// TIA Portal V20 export
FUNCTION "03 T10 LANT Aux" : Void   // FC1393, LAD
TITLE = AUXILIARIES
{ S7_Optimized_Access := 'TRUE' }
// stored: AutoNumber false, SetENOAutomatically false
   VAR_TEMP
      Aux_OS : Bool;
      Aux_sup : Real;
      Aux_inf : Real;
      Aux_DInt : DInt;
      Aux_Real : Real;
   END_VAR
   VAR CONSTANT
      "Max differenza L tubi" : Real := 500.0;
   END_VAR
   VAR_TEMP   // added for the SCL form of the ladder/FBD networks
      _w1 : Bool;
      _w2 : Bool;
      _w3 : Bool;
   END_VAR
BEGIN

REGION Network 1: =========== MEMORIES ===========
END_REGION

REGION Network 2: Piece presence
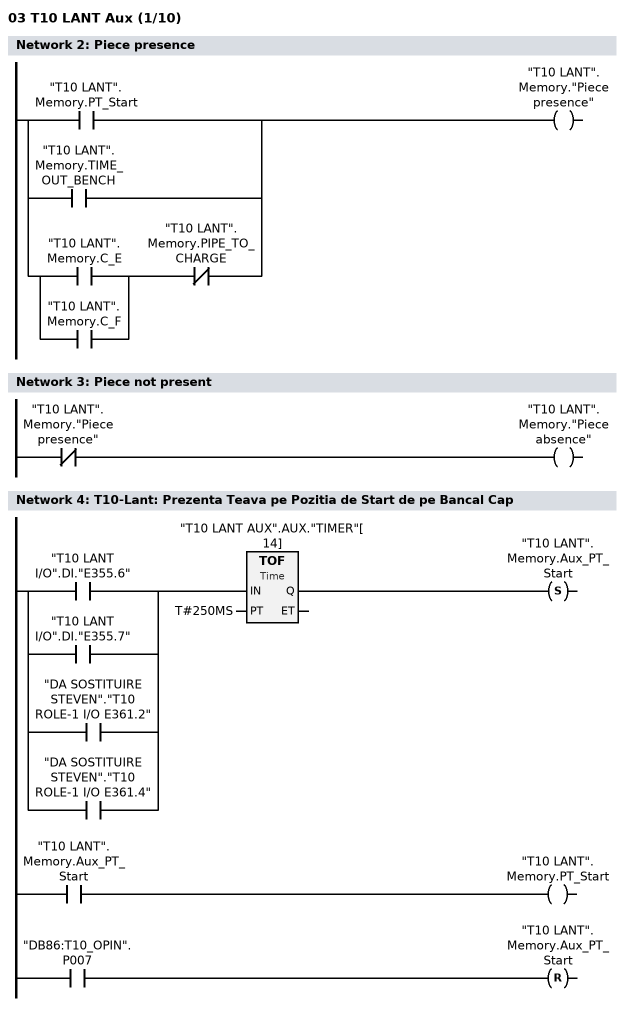
   RUNG wire#powerrail
      Contact( "T10 LANT".Memory.PT_Start )
      wire#w1
      Coil( "T10 LANT".Memory."Piece presence" )
   END_RUNG
   RUNG wire#powerrail
      Contact( "T10 LANT".Memory.TIME_OUT_BENCH )
   END_RUNG wire#w1
   RUNG wire#powerrail
      Contact( "T10 LANT".Memory.C_E )
      wire#w2
      I_Contact( "T10 LANT".Memory.PIPE_TO_CHARGE )
   END_RUNG wire#w1
   RUNG wire#powerrail
      Contact( "T10 LANT".Memory.C_F )
   END_RUNG wire#w2
   // the same network as SCL:
   "T10 LANT".Memory."Piece presence" := "T10 LANT".Memory.PT_Start OR "T10 LANT".Memory.TIME_OUT_BENCH OR (("T10 LANT".Memory.C_E OR "T10 LANT".Memory.C_F) AND NOT "T10 LANT".Memory.PIPE_TO_CHARGE);
END_REGION

REGION Network 3: Piece not present
   RUNG wire#powerrail
      I_Contact( "T10 LANT".Memory."Piece presence" )
      Coil( "T10 LANT".Memory."Piece absence" )
   END_RUNG
   // the same network as SCL:
   "T10 LANT".Memory."Piece absence" := NOT "T10 LANT".Memory."Piece presence";
END_REGION

REGION Network 4: T10-Lant: Prezenta Teava pe Pozitia de Start de pe Bancal Cap
   RUNG wire#powerrail
      Contact( "T10 LANT I/O".DI."E355.6" )
      wire#w1
      { S7_Templates := "time_type := Time" } "T10 LANT AUX".AUX."TIMER"[14].TOF(pt := T#250MS, et =>)
      S_Coil( "T10 LANT".Memory.Aux_PT_Start )
   END_RUNG
   RUNG wire#powerrail
      Contact( "T10 LANT I/O".DI."E355.7" )
   END_RUNG wire#w1
   RUNG wire#powerrail
      Contact( "DA SOSTITUIRE STEVEN"."T10 ROLE-1 I/O E361.2" )
   END_RUNG wire#w1
   RUNG wire#powerrail
      Contact( "DA SOSTITUIRE STEVEN"."T10 ROLE-1 I/O E361.4" )
   END_RUNG wire#w1
   RUNG wire#powerrail
      Contact( "T10 LANT".Memory.Aux_PT_Start )
      Coil( "T10 LANT".Memory.PT_Start )
   END_RUNG
   RUNG wire#powerrail
      Contact( "DB86:T10_OPIN".P007 )
      R_Coil( "T10 LANT".Memory.Aux_PT_Start )
   END_RUNG
   // the same network as SCL:
   "T10 LANT AUX".AUX."TIMER"[14].TOF(IN := "T10 LANT I/O".DI."E355.6" OR "T10 LANT I/O".DI."E355.7" OR "DA SOSTITUIRE STEVEN"."T10 ROLE-1 I/O E361.2" OR "DA SOSTITUIRE STEVEN"."T10 ROLE-1 I/O E361.4",
                           PT := T#250MS);
   IF "T10 LANT AUX".AUX."TIMER"[14].Q THEN "T10 LANT".Memory.Aux_PT_Start := TRUE; END_IF;
   "T10 LANT".Memory.PT_Start := "T10 LANT".Memory.Aux_PT_Start;
   IF "DB86:T10_OPIN".P007 THEN "T10 LANT".Memory.Aux_PT_Start := FALSE; END_IF;
END_REGION

REGION Network 5: T10-Lant: Prezenta Teava pe Pozitia de 'Incetinire' de pe Bancal
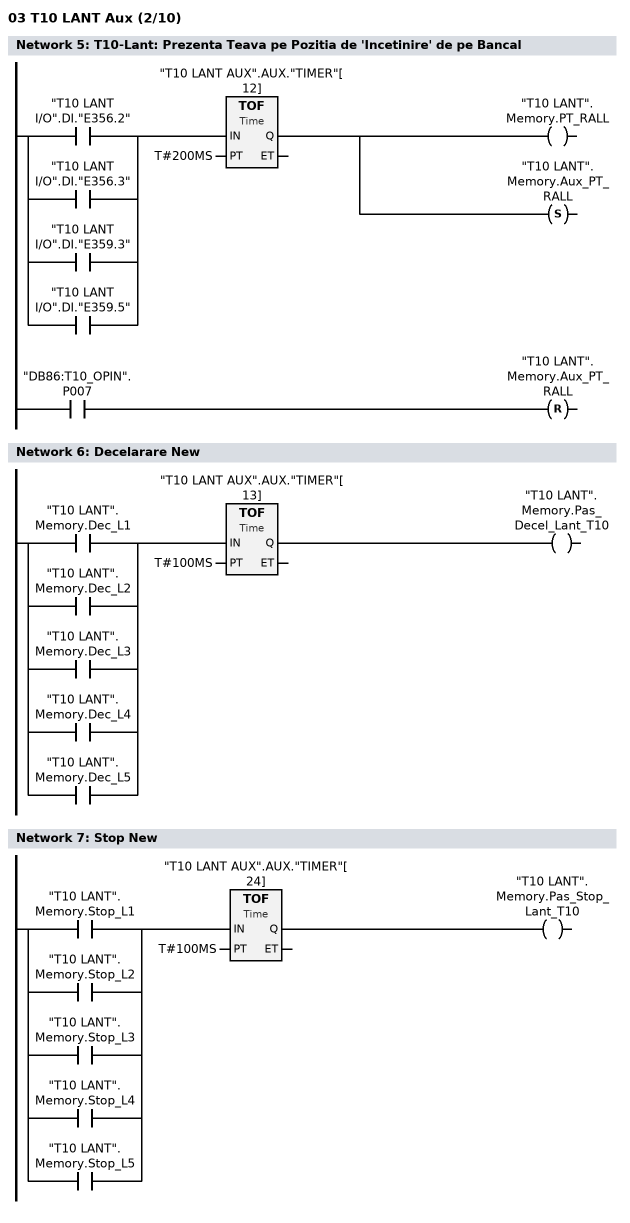
   RUNG wire#powerrail
      Contact( "T10 LANT I/O".DI."E356.2" )
      wire#w1
      { S7_Templates := "time_type := Time" } "T10 LANT AUX".AUX."TIMER"[12].TOF(pt := T#200MS, et =>)
      wire#w2
      Coil( "T10 LANT".Memory.PT_RALL )
   END_RUNG
   RUNG wire#powerrail
      Contact( "T10 LANT I/O".DI."E356.3" )
   END_RUNG wire#w1
   RUNG wire#powerrail
      Contact( "T10 LANT I/O".DI."E359.3" )
   END_RUNG wire#w1
   RUNG wire#powerrail
      Contact( "T10 LANT I/O".DI."E359.5" )
   END_RUNG wire#w1
   RUNG wire#w2
      S_Coil( "T10 LANT".Memory.Aux_PT_RALL )
   END_RUNG
   RUNG wire#powerrail
      Contact( "DB86:T10_OPIN".P007 )
      R_Coil( "T10 LANT".Memory.Aux_PT_RALL )
   END_RUNG
   // the same network as SCL:
   "T10 LANT AUX".AUX."TIMER"[12].TOF(IN := "T10 LANT I/O".DI."E356.2" OR "T10 LANT I/O".DI."E356.3" OR "T10 LANT I/O".DI."E359.3" OR "T10 LANT I/O".DI."E359.5",
                           PT := T#200MS);
   "T10 LANT".Memory.PT_RALL := "T10 LANT AUX".AUX."TIMER"[12].Q;
   IF "T10 LANT AUX".AUX."TIMER"[12].Q THEN "T10 LANT".Memory.Aux_PT_RALL := TRUE; END_IF;
   IF "DB86:T10_OPIN".P007 THEN "T10 LANT".Memory.Aux_PT_RALL := FALSE; END_IF;
END_REGION

REGION Network 6: Decelarare New
   RUNG wire#powerrail
      Contact( "T10 LANT".Memory.Dec_L1 )
      wire#w1
      { S7_Templates := "time_type := Time" } "T10 LANT AUX".AUX."TIMER"[13].TOF(pt := T#100MS, et =>)
      Coil( "T10 LANT".Memory.Pas_Decel_Lant_T10 )
   END_RUNG
   RUNG wire#powerrail
      Contact( "T10 LANT".Memory.Dec_L2 )
   END_RUNG wire#w1
   RUNG wire#powerrail
      Contact( "T10 LANT".Memory.Dec_L3 )
   END_RUNG wire#w1
   RUNG wire#powerrail
      Contact( "T10 LANT".Memory.Dec_L4 )
   END_RUNG wire#w1
   RUNG wire#powerrail
      Contact( "T10 LANT".Memory.Dec_L5 )
   END_RUNG wire#w1
   // the same network as SCL:
   "T10 LANT AUX".AUX."TIMER"[13].TOF(IN := "T10 LANT".Memory.Dec_L1 OR "T10 LANT".Memory.Dec_L2 OR "T10 LANT".Memory.Dec_L3 OR "T10 LANT".Memory.Dec_L4 OR "T10 LANT".Memory.Dec_L5,
                           PT := T#100MS);
   "T10 LANT".Memory.Pas_Decel_Lant_T10 := "T10 LANT AUX".AUX."TIMER"[13].Q;
END_REGION

REGION Network 7: Stop New
   RUNG wire#powerrail
      Contact( "T10 LANT".Memory.Stop_L1 )
      wire#w1
      { S7_Templates := "time_type := Time" } "T10 LANT AUX".AUX."TIMER"[24].TOF(pt := T#100MS, et =>)
      Coil( "T10 LANT".Memory.Pas_Stop_Lant_T10 )
   END_RUNG
   RUNG wire#powerrail
      Contact( "T10 LANT".Memory.Stop_L2 )
   END_RUNG wire#w1
   RUNG wire#powerrail
      Contact( "T10 LANT".Memory.Stop_L3 )
   END_RUNG wire#w1
   RUNG wire#powerrail
      Contact( "T10 LANT".Memory.Stop_L4 )
   END_RUNG wire#w1
   RUNG wire#powerrail
      Contact( "T10 LANT".Memory.Stop_L5 )
   END_RUNG wire#w1
   // the same network as SCL:
   "T10 LANT AUX".AUX."TIMER"[24].TOF(IN := "T10 LANT".Memory.Stop_L1 OR "T10 LANT".Memory.Stop_L2 OR "T10 LANT".Memory.Stop_L3 OR "T10 LANT".Memory.Stop_L4 OR "T10 LANT".Memory.Stop_L5,
                           PT := T#100MS);
   "T10 LANT".Memory.Pas_Stop_Lant_T10 := "T10 LANT AUX".AUX."TIMER"[24].Q;
END_REGION

REGION Network 8: T10-Lant: LAnt in Pozitia 'Pas'
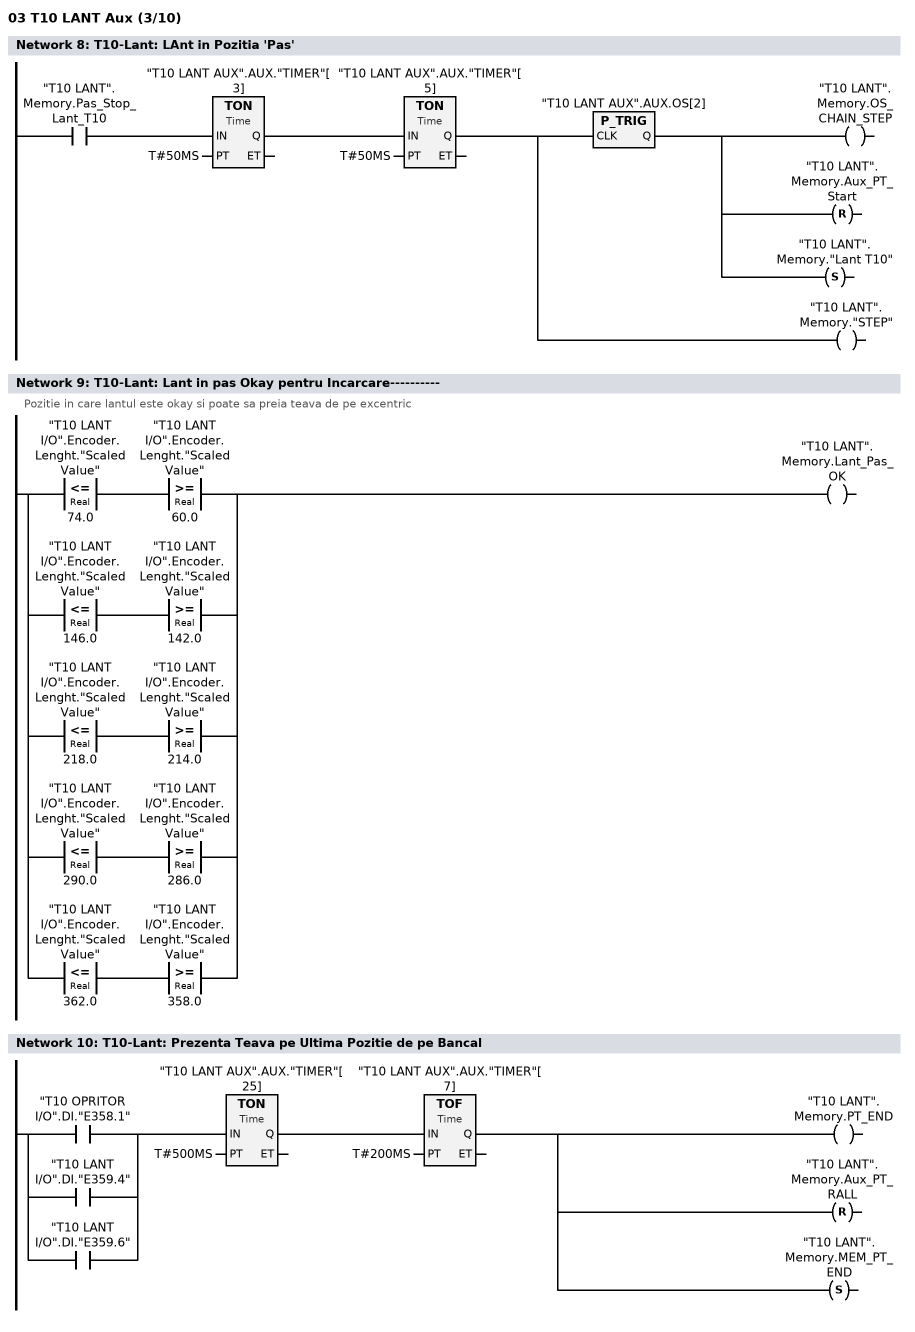
   RUNG wire#powerrail
      Contact( "T10 LANT".Memory.Pas_Stop_Lant_T10 )
      { S7_Templates := "time_type := Time" } "T10 LANT AUX".AUX."TIMER"[3].TON(pt := T#50MS, et =>)
      { S7_Templates := "time_type := Time" } "T10 LANT AUX".AUX."TIMER"[5].TON(pt := T#50MS, et =>)
      wire#w1
      P_Trig( "T10 LANT AUX".AUX.OS[2] )
      wire#w2
      Coil( "T10 LANT".Memory.OS_CHAIN_STEP )
   END_RUNG
   RUNG wire#w2
      R_Coil( "T10 LANT".Memory.Aux_PT_Start )
   END_RUNG
   RUNG wire#w2
      S_Coil( "T10 LANT".Memory."Lant T10" )
   END_RUNG
   RUNG wire#w1
      Coil( "T10 LANT".Memory."STEP" )
   END_RUNG
   // the same network as SCL:
   "T10 LANT AUX".AUX."TIMER"[3].TON(IN := "T10 LANT".Memory.Pas_Stop_Lant_T10, PT := T#50MS);
   "T10 LANT AUX".AUX."TIMER"[5].TON(IN := "T10 LANT AUX".AUX."TIMER"[3].Q, PT := T#50MS);
   #_w1 := "T10 LANT AUX".AUX."TIMER"[5].Q AND NOT "T10 LANT AUX".AUX.OS[2];   // rising edge
   "T10 LANT AUX".AUX.OS[2] := "T10 LANT AUX".AUX."TIMER"[5].Q;
   "T10 LANT".Memory.OS_CHAIN_STEP := #_w1;
   IF #_w1 THEN
       "T10 LANT".Memory.Aux_PT_Start := FALSE;
       "T10 LANT".Memory."Lant T10" := TRUE;
   END_IF;
   "T10 LANT".Memory."STEP" := "T10 LANT AUX".AUX."TIMER"[5].Q;
END_REGION

REGION Network 9: T10-Lant: Lant in pas Okay pentru Incarcare----------
   // Pozitie in care lantul este okay si poate sa preia teava de pe excentric
   RUNG wire#powerrail
      { S7_Templates := "SrcType := Real" } LE_Contact(in1 := "T10 LANT I/O".Encoder.Lenght."Scaled Value", in2 := 74.0)
      { S7_Templates := "SrcType := Real" } GE_Contact(in1 := "T10 LANT I/O".Encoder.Lenght."Scaled Value", in2 := 60.0)
      wire#w1
      Coil( "T10 LANT".Memory.Lant_Pas_OK )
   END_RUNG
   RUNG wire#powerrail
      { S7_Templates := "SrcType := Real" } LE_Contact(in1 := "T10 LANT I/O".Encoder.Lenght."Scaled Value", in2 := 146.0)
      { S7_Templates := "SrcType := Real" } GE_Contact(in1 := "T10 LANT I/O".Encoder.Lenght."Scaled Value", in2 := 142.0)
   END_RUNG wire#w1
   RUNG wire#powerrail
      { S7_Templates := "SrcType := Real" } LE_Contact(in1 := "T10 LANT I/O".Encoder.Lenght."Scaled Value", in2 := 218.0)
      { S7_Templates := "SrcType := Real" } GE_Contact(in1 := "T10 LANT I/O".Encoder.Lenght."Scaled Value", in2 := 214.0)
   END_RUNG wire#w1
   RUNG wire#powerrail
      { S7_Templates := "SrcType := Real" } LE_Contact(in1 := "T10 LANT I/O".Encoder.Lenght."Scaled Value", in2 := 290.0)
      { S7_Templates := "SrcType := Real" } GE_Contact(in1 := "T10 LANT I/O".Encoder.Lenght."Scaled Value", in2 := 286.0)
   END_RUNG wire#w1
   RUNG wire#powerrail
      { S7_Templates := "SrcType := Real" } LE_Contact(in1 := "T10 LANT I/O".Encoder.Lenght."Scaled Value", in2 := 362.0)
      { S7_Templates := "SrcType := Real" } GE_Contact(in1 := "T10 LANT I/O".Encoder.Lenght."Scaled Value", in2 := 358.0)
   END_RUNG wire#w1
   // the same network as SCL:
   "T10 LANT".Memory.Lant_Pas_OK := (("T10 LANT I/O".Encoder.Lenght."Scaled Value" <= 74.0) AND ("T10 LANT I/O".Encoder.Lenght."Scaled Value" >= 60.0)) OR (("T10 LANT I/O".Encoder.Lenght."Scaled Value" <= 146.0) AND ("T10 LANT I/O".Encoder.Lenght."Scaled Value" >= 142.0)) OR (("T10 LANT I/O".Encoder.Lenght."Scaled Value" <= 218.0) AND ("T10 LANT I/O".Encoder.Lenght."Scaled Value" >= 214.0)) OR (("T10 LANT I/O".Encoder.Lenght."Scaled Value" <= 290.0) AND ("T10 LANT I/O".Encoder.Lenght."Scaled Value" >= 286.0)) OR (("T10 LANT I/O".Encoder.Lenght."Scaled Value" <= 362.0) AND ("T10 LANT I/O".Encoder.Lenght."Scaled Value" >= 358.0));
END_REGION

REGION Network 10: T10-Lant: Prezenta Teava pe Ultima Pozitie de pe Bancal
   RUNG wire#powerrail
      Contact( "T10 OPRITOR I/O".DI."E358.1" )
      wire#w1
      { S7_Templates := "time_type := Time" } "T10 LANT AUX".AUX."TIMER"[25].TON(pt := T#500MS, et =>)
      { S7_Templates := "time_type := Time" } "T10 LANT AUX".AUX."TIMER"[7].TOF(pt := T#200MS, et =>)
      wire#w2
      Coil( "T10 LANT".Memory.PT_END )
   END_RUNG
   RUNG wire#powerrail
      Contact( "T10 LANT I/O".DI."E359.4" )
   END_RUNG wire#w1
   RUNG wire#powerrail
      Contact( "T10 LANT I/O".DI."E359.6" )
   END_RUNG wire#w1
   RUNG wire#w2
      R_Coil( "T10 LANT".Memory.Aux_PT_RALL )
   END_RUNG
   RUNG wire#w2
      S_Coil( "T10 LANT".Memory.MEM_PT_END )
   END_RUNG
   // the same network as SCL:
   "T10 LANT AUX".AUX."TIMER"[25].TON(IN := "T10 OPRITOR I/O".DI."E358.1" OR "T10 LANT I/O".DI."E359.4" OR "T10 LANT I/O".DI."E359.6",
                           PT := T#500MS);
   "T10 LANT AUX".AUX."TIMER"[7].TOF(IN := "T10 LANT AUX".AUX."TIMER"[25].Q, PT := T#200MS);
   "T10 LANT".Memory.PT_END := "T10 LANT AUX".AUX."TIMER"[7].Q;
   IF "T10 LANT AUX".AUX."TIMER"[7].Q THEN
       "T10 LANT".Memory.Aux_PT_RALL := FALSE;
       "T10 LANT".Memory.MEM_PT_END := TRUE;
   END_IF;
END_REGION

REGION Network 11: T10-Lant: TRK: Prezenta Teava pe Pozitia 'Incetinire' pe Bancal
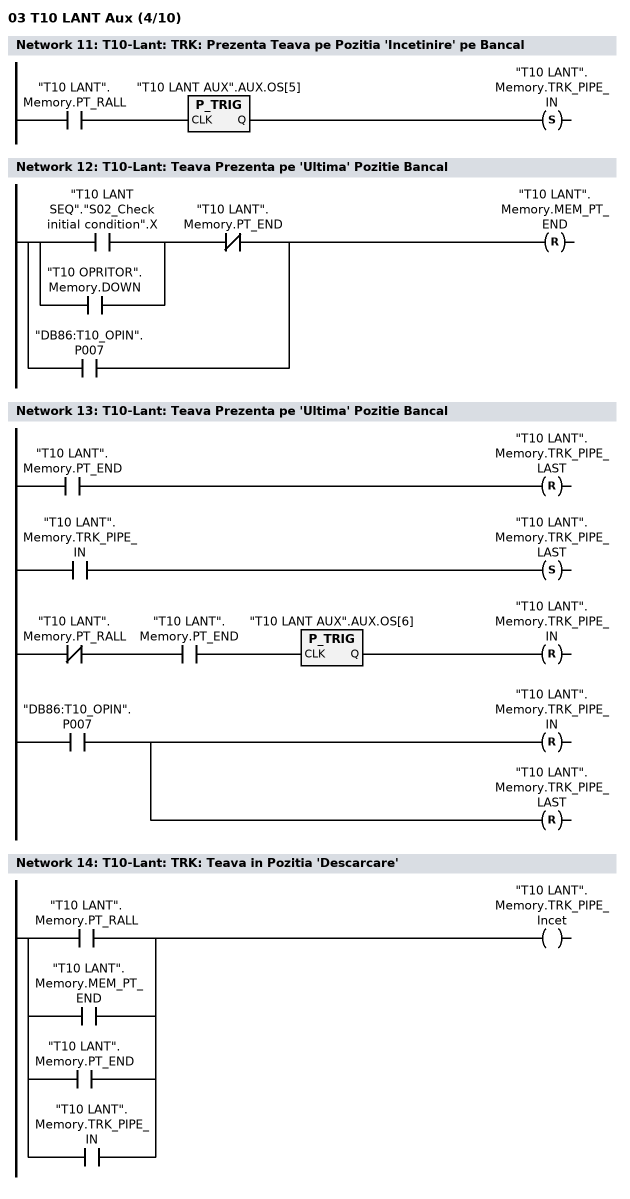
   RUNG wire#powerrail
      Contact( "T10 LANT".Memory.PT_RALL )
      P_Trig( "T10 LANT AUX".AUX.OS[5] )
      S_Coil( "T10 LANT".Memory.TRK_PIPE_IN )
   END_RUNG
   // the same network as SCL:
   #_w1 := "T10 LANT".Memory.PT_RALL AND NOT "T10 LANT AUX".AUX.OS[5];   // rising edge
   "T10 LANT AUX".AUX.OS[5] := "T10 LANT".Memory.PT_RALL;
   IF #_w1 THEN "T10 LANT".Memory.TRK_PIPE_IN := TRUE; END_IF;
END_REGION

REGION Network 12: T10-Lant: Teava Prezenta pe 'Ultima' Pozitie Bancal
   RUNG wire#powerrail
      Contact( "T10 LANT SEQ"."S02_Check initial condition".X )
      wire#w1
      I_Contact( "T10 LANT".Memory.PT_END )
      wire#w2
      R_Coil( "T10 LANT".Memory.MEM_PT_END )
   END_RUNG
   RUNG wire#powerrail
      Contact( "T10 OPRITOR".Memory.DOWN )
   END_RUNG wire#w1
   RUNG wire#powerrail
      Contact( "DB86:T10_OPIN".P007 )
   END_RUNG wire#w2
   // the same network as SCL:
   IF (("T10 LANT SEQ"."S02_Check initial condition".X OR "T10 OPRITOR".Memory.DOWN) AND NOT "T10 LANT".Memory.PT_END) OR "DB86:T10_OPIN".P007 THEN
       "T10 LANT".Memory.MEM_PT_END := FALSE;
   END_IF;
END_REGION

REGION Network 13: T10-Lant: Teava Prezenta pe 'Ultima' Pozitie Bancal
   RUNG wire#powerrail
      Contact( "T10 LANT".Memory.PT_END )
      R_Coil( "T10 LANT".Memory.TRK_PIPE_LAST )
   END_RUNG
   RUNG wire#powerrail
      Contact( "T10 LANT".Memory.TRK_PIPE_IN )
      S_Coil( "T10 LANT".Memory.TRK_PIPE_LAST )
   END_RUNG
   RUNG wire#powerrail
      I_Contact( "T10 LANT".Memory.PT_RALL )
      Contact( "T10 LANT".Memory.PT_END )
      P_Trig( "T10 LANT AUX".AUX.OS[6] )
      R_Coil( "T10 LANT".Memory.TRK_PIPE_IN )
   END_RUNG
   RUNG wire#powerrail
      Contact( "DB86:T10_OPIN".P007 )
      wire#w1
      R_Coil( "T10 LANT".Memory.TRK_PIPE_IN )
   END_RUNG
   RUNG wire#w1
      R_Coil( "T10 LANT".Memory.TRK_PIPE_LAST )
   END_RUNG
   // the same network as SCL:
   IF "T10 LANT".Memory.PT_END THEN "T10 LANT".Memory.TRK_PIPE_LAST := FALSE; END_IF;
   IF "T10 LANT".Memory.TRK_PIPE_IN THEN "T10 LANT".Memory.TRK_PIPE_LAST := TRUE; END_IF;
   #_w1 := NOT "T10 LANT".Memory.PT_RALL AND "T10 LANT".Memory.PT_END;
   #_w2 := #_w1 AND NOT "T10 LANT AUX".AUX.OS[6];   // rising edge
   "T10 LANT AUX".AUX.OS[6] := #_w1;
   IF #_w2 THEN "T10 LANT".Memory.TRK_PIPE_IN := FALSE; END_IF;
   IF "DB86:T10_OPIN".P007 THEN
       "T10 LANT".Memory.TRK_PIPE_IN := FALSE;
       "T10 LANT".Memory.TRK_PIPE_LAST := FALSE;
   END_IF;
END_REGION

REGION Network 14: T10-Lant: TRK: Teava in Pozitia 'Descarcare'
   RUNG wire#powerrail
      Contact( "T10 LANT".Memory.PT_RALL )
      wire#w1
      Coil( "T10 LANT".Memory.TRK_PIPE_Incet )
   END_RUNG
   RUNG wire#powerrail
      Contact( "T10 LANT".Memory.MEM_PT_END )
   END_RUNG wire#w1
   RUNG wire#powerrail
      Contact( "T10 LANT".Memory.PT_END )
   END_RUNG wire#w1
   RUNG wire#powerrail
      Contact( "T10 LANT".Memory.TRK_PIPE_IN )
   END_RUNG wire#w1
   // the same network as SCL:
   "T10 LANT".Memory.TRK_PIPE_Incet := "T10 LANT".Memory.PT_RALL OR "T10 LANT".Memory.MEM_PT_END OR "T10 LANT".Memory.PT_END OR "T10 LANT".Memory.TRK_PIPE_IN;
END_REGION

REGION Network 15: T10-Lant: Teava Pregatita pt. 'Incarcare'
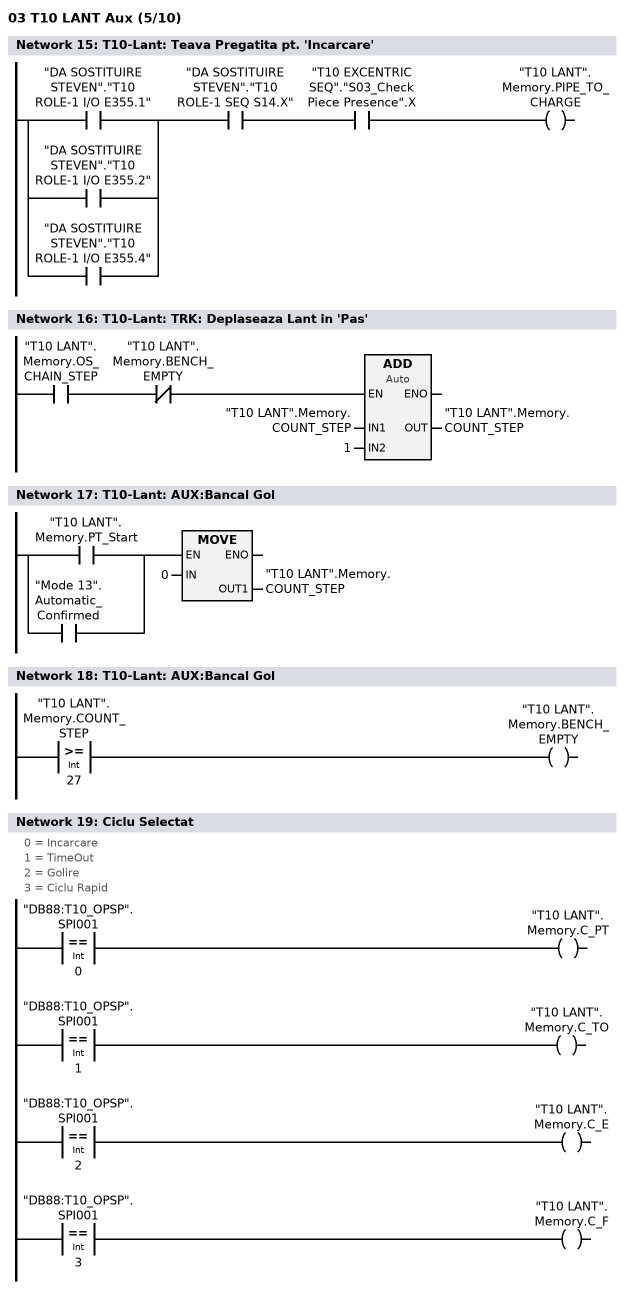
   RUNG wire#powerrail
      Contact( "DA SOSTITUIRE STEVEN"."T10 ROLE-1 I/O E355.1" )
      wire#w1
      Contact( "DA SOSTITUIRE STEVEN"."T10 ROLE-1 SEQ S14.X" )
      Contact( "T10 EXCENTRIC SEQ"."S03_Check Piece Presence".X )
      Coil( "T10 LANT".Memory.PIPE_TO_CHARGE )
   END_RUNG
   RUNG wire#powerrail
      Contact( "DA SOSTITUIRE STEVEN"."T10 ROLE-1 I/O E355.2" )
   END_RUNG wire#w1
   RUNG wire#powerrail
      Contact( "DA SOSTITUIRE STEVEN"."T10 ROLE-1 I/O E355.4" )
   END_RUNG wire#w1
   // the same network as SCL:
   "T10 LANT".Memory.PIPE_TO_CHARGE := ("DA SOSTITUIRE STEVEN"."T10 ROLE-1 I/O E355.1" OR "DA SOSTITUIRE STEVEN"."T10 ROLE-1 I/O E355.2" OR "DA SOSTITUIRE STEVEN"."T10 ROLE-1 I/O E355.4") AND "DA SOSTITUIRE STEVEN"."T10 ROLE-1 SEQ S14.X" AND "T10 EXCENTRIC SEQ"."S03_Check Piece Presence".X;
END_REGION

REGION Network 16: T10-Lant: TRK: Deplaseaza Lant in 'Pas'
   RUNG wire#powerrail
      Contact( "T10 LANT".Memory.OS_CHAIN_STEP )
      I_Contact( "T10 LANT".Memory.BENCH_EMPTY )
      Add(in1 := "T10 LANT".Memory.COUNT_STEP, in2 := 1, out => "T10 LANT".Memory.COUNT_STEP)
   END_RUNG
   // the same network as SCL:
   IF "T10 LANT".Memory.OS_CHAIN_STEP AND NOT "T10 LANT".Memory.BENCH_EMPTY THEN
       "T10 LANT".Memory.COUNT_STEP := "T10 LANT".Memory.COUNT_STEP + 1;
   END_IF;
END_REGION

REGION Network 17: T10-Lant: AUX:Bancal Gol
   RUNG wire#powerrail
      Contact( "T10 LANT".Memory.PT_Start )
      wire#w1
      Move(in := 0, out1 => "T10 LANT".Memory.COUNT_STEP)
   END_RUNG
   RUNG wire#powerrail
      Contact( "Mode 13".Automatic_Confirmed )
   END_RUNG wire#w1
   // the same network as SCL:
   IF "T10 LANT".Memory.PT_Start OR "Mode 13".Automatic_Confirmed THEN
       "T10 LANT".Memory.COUNT_STEP := 0;
   END_IF;
END_REGION

REGION Network 18: T10-Lant: AUX:Bancal Gol
   RUNG wire#powerrail
      { S7_Templates := "SrcType := Int" } GE_Contact(in1 := "T10 LANT".Memory.COUNT_STEP, in2 := 27)
      Coil( "T10 LANT".Memory.BENCH_EMPTY )
   END_RUNG
   // the same network as SCL:
   "T10 LANT".Memory.BENCH_EMPTY := "T10 LANT".Memory.COUNT_STEP >= 27;
END_REGION

REGION Network 19: Ciclu Selectat
   // 0 = Incarcare 
   // 1 = TimeOut
   // 2 = Golire
   // 3 = Ciclu Rapid
   RUNG wire#powerrail
      { S7_Templates := "SrcType := Int" } EQ_Contact(in1 := "DB88:T10_OPSP".SPI001, in2 := 0)
      Coil( "T10 LANT".Memory.C_PT )
   END_RUNG
   RUNG wire#powerrail
      { S7_Templates := "SrcType := Int" } EQ_Contact(in1 := "DB88:T10_OPSP".SPI001, in2 := 1)
      Coil( "T10 LANT".Memory.C_TO )
   END_RUNG
   RUNG wire#powerrail
      { S7_Templates := "SrcType := Int" } EQ_Contact(in1 := "DB88:T10_OPSP".SPI001, in2 := 2)
      Coil( "T10 LANT".Memory.C_E )
   END_RUNG
   RUNG wire#powerrail
      { S7_Templates := "SrcType := Int" } EQ_Contact(in1 := "DB88:T10_OPSP".SPI001, in2 := 3)
      Coil( "T10 LANT".Memory.C_F )
   END_RUNG
   // the same network as SCL:
   "T10 LANT".Memory.C_PT := "DB88:T10_OPSP".SPI001 = 0;
   "T10 LANT".Memory.C_TO := "DB88:T10_OPSP".SPI001 = 1;
   "T10 LANT".Memory.C_E := "DB88:T10_OPSP".SPI001 = 2;
   "T10 LANT".Memory.C_F := "DB88:T10_OPSP".SPI001 = 3;
END_REGION

REGION Network 20: Lant T10 Pasi
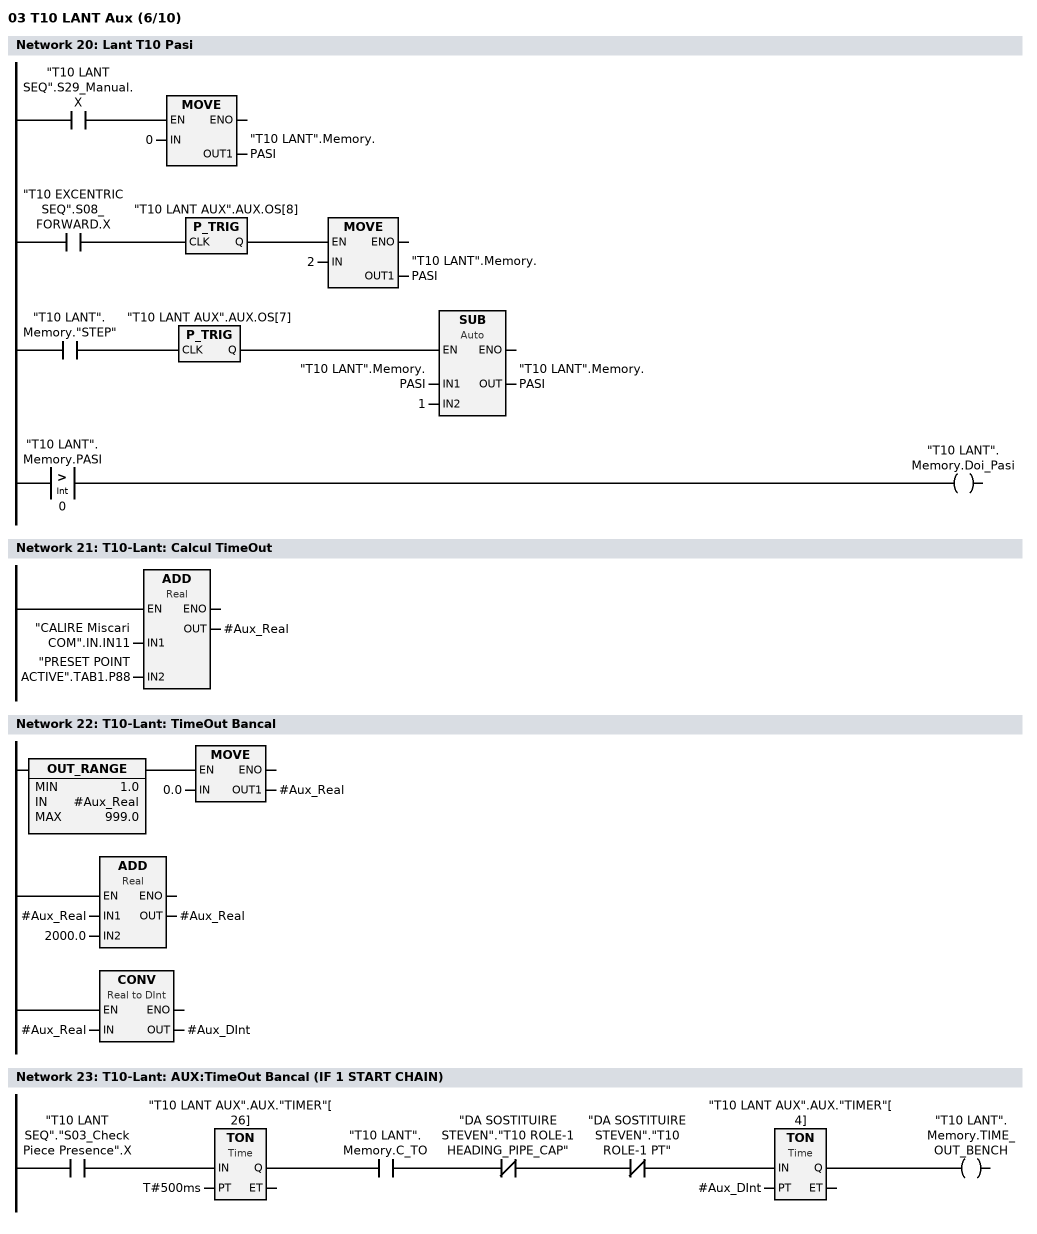
   RUNG wire#powerrail
      Contact( "T10 LANT SEQ".S29_Manual.X )
      Move(in := 0, out1 => "T10 LANT".Memory.PASI)
   END_RUNG
   RUNG wire#powerrail
      Contact( "T10 EXCENTRIC SEQ".S08_FORWARD.X )
      P_Trig( "T10 LANT AUX".AUX.OS[8] )
      Move(in := 2, out1 => "T10 LANT".Memory.PASI)
   END_RUNG
   RUNG wire#powerrail
      Contact( "T10 LANT".Memory."STEP" )
      P_Trig( "T10 LANT AUX".AUX.OS[7] )
      Sub(in1 := "T10 LANT".Memory.PASI, in2 := 1, out => "T10 LANT".Memory.PASI)
   END_RUNG
   RUNG wire#powerrail
      { S7_Templates := "SrcType := Int" } GT_Contact(in1 := "T10 LANT".Memory.PASI, in2 := 0)
      Coil( "T10 LANT".Memory.Doi_Pasi )
   END_RUNG
   // the same network as SCL:
   IF "T10 LANT SEQ".S29_Manual.X THEN "T10 LANT".Memory.PASI := 0; END_IF;
   #_w1 := "T10 EXCENTRIC SEQ".S08_FORWARD.X AND NOT "T10 LANT AUX".AUX.OS[8];   // rising edge
   "T10 LANT AUX".AUX.OS[8] := "T10 EXCENTRIC SEQ".S08_FORWARD.X;
   IF #_w1 THEN "T10 LANT".Memory.PASI := 2; END_IF;
   #_w2 := "T10 LANT".Memory."STEP" AND NOT "T10 LANT AUX".AUX.OS[7];   // rising edge
   "T10 LANT AUX".AUX.OS[7] := "T10 LANT".Memory."STEP";
   IF #_w2 THEN "T10 LANT".Memory.PASI := "T10 LANT".Memory.PASI - 1; END_IF;
   "T10 LANT".Memory.Doi_Pasi := "T10 LANT".Memory.PASI > 0;
END_REGION

REGION Network 21: T10-Lant: Calcul TimeOut
   RUNG wire#powerrail
      { S7_Templates := "SrcType := Real" } Add(in1 := "CALIRE Miscari COM".IN.IN11, in2 := "PRESET POINT ACTIVE".TAB1.P88, out => #Aux_Real)
   END_RUNG
   // the same network as SCL:
   #Aux_Real := "CALIRE Miscari COM".IN.IN11 + "PRESET POINT ACTIVE".TAB1.P88;
END_REGION

REGION Network 22: T10-Lant: TimeOut Bancal
   IF (#Aux_Real < 1.0) OR (#Aux_Real > 999.0) THEN #Aux_Real := 0.0; END_IF;
   #Aux_Real := #Aux_Real + 2000.0;
   #Aux_DInt := REAL_TO_DINT(#Aux_Real);
END_REGION

REGION Network 23: T10-Lant: AUX:TimeOut Bancal (IF 1 START CHAIN)
   RUNG wire#powerrail
      Contact( "T10 LANT SEQ"."S03_Check Piece Presence".X )
      { S7_Templates := "time_type := Time" } "T10 LANT AUX".AUX."TIMER"[26].TON(pt := T#500ms, et =>)
      Contact( "T10 LANT".Memory.C_TO )
      I_Contact( "DA SOSTITUIRE STEVEN"."T10 ROLE-1 HEADING_PIPE_CAP" )
      I_Contact( "DA SOSTITUIRE STEVEN"."T10 ROLE-1 PT" )
      { S7_Templates := "time_type := Time" } "T10 LANT AUX".AUX."TIMER"[4].TON(pt := #Aux_DInt, et =>)
      Coil( "T10 LANT".Memory.TIME_OUT_BENCH )
   END_RUNG
   // the same network as SCL:
   "T10 LANT AUX".AUX."TIMER"[26].TON(IN := "T10 LANT SEQ"."S03_Check Piece Presence".X, PT := T#500ms);
   "T10 LANT AUX".AUX."TIMER"[4].TON(IN := "T10 LANT AUX".AUX."TIMER"[26].Q AND "T10 LANT".Memory.C_TO AND NOT "DA SOSTITUIRE STEVEN"."T10 ROLE-1 HEADING_PIPE_CAP" AND NOT "DA SOSTITUIRE STEVEN"."T10 ROLE-1 PT",
                           PT := #Aux_DInt);
   "T10 LANT".Memory.TIME_OUT_BENCH := "T10 LANT AUX".AUX."TIMER"[4].Q;
END_REGION

REGION Network 24: Memories - Local Auto Stop
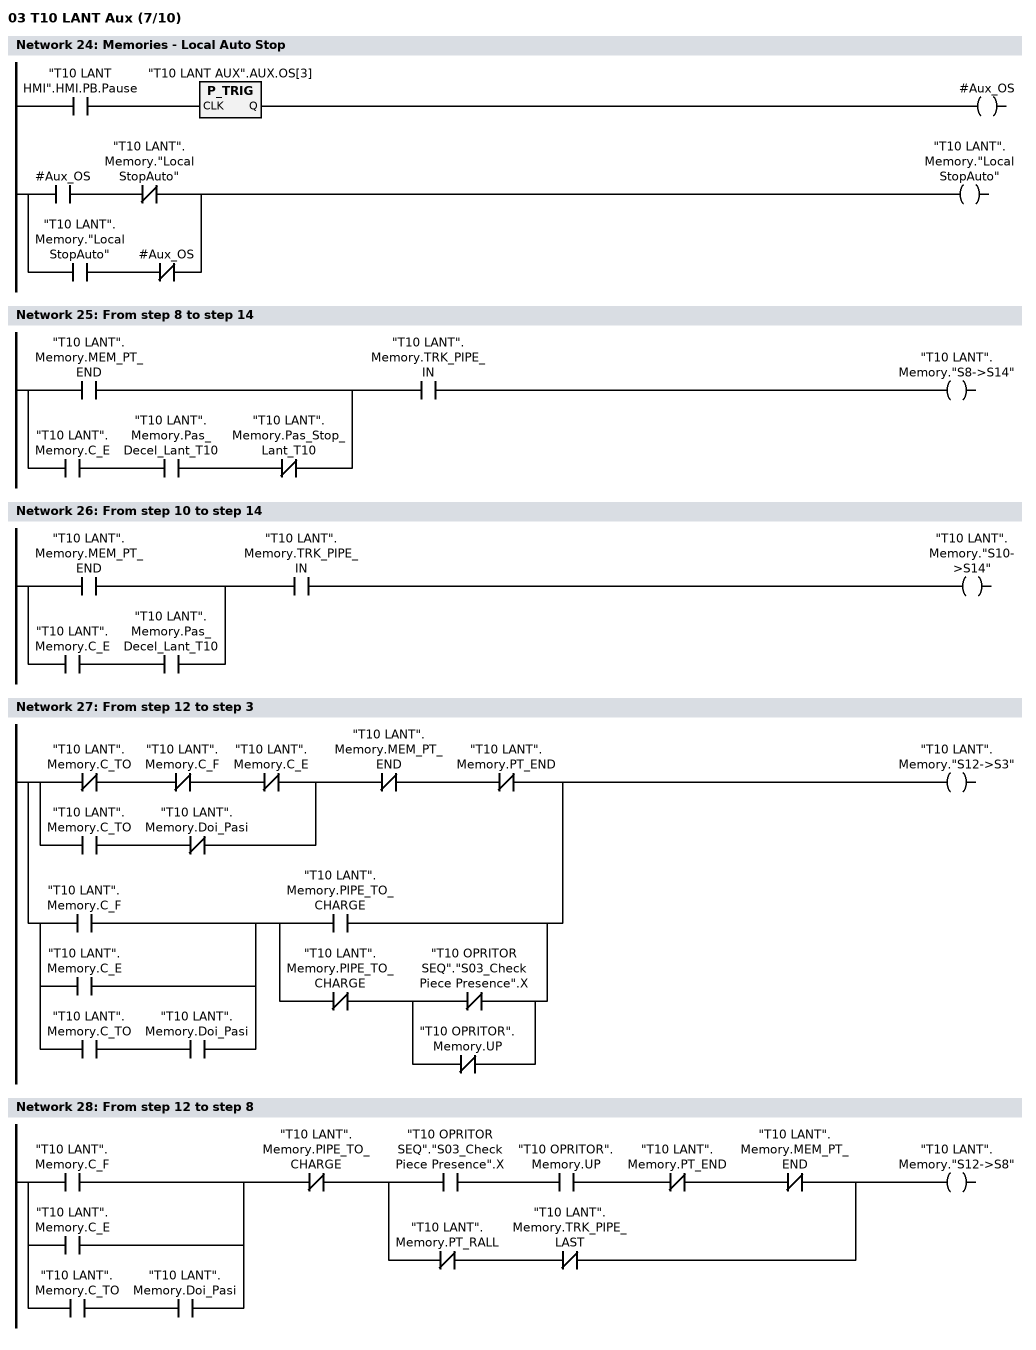
   RUNG wire#powerrail
      Contact( "T10 LANT HMI".HMI.PB.Pause )
      P_Trig( "T10 LANT AUX".AUX.OS[3] )
      Coil( #Aux_OS )
   END_RUNG
   RUNG wire#powerrail
      Contact( #Aux_OS )
      I_Contact( "T10 LANT".Memory."Local StopAuto" )
      wire#w1
      Coil( "T10 LANT".Memory."Local StopAuto" )
   END_RUNG
   RUNG wire#powerrail
      Contact( "T10 LANT".Memory."Local StopAuto" )
      I_Contact( #Aux_OS )
   END_RUNG wire#w1
   // the same network as SCL:
   #_w1 := "T10 LANT HMI".HMI.PB.Pause AND NOT "T10 LANT AUX".AUX.OS[3];   // rising edge
   "T10 LANT AUX".AUX.OS[3] := "T10 LANT HMI".HMI.PB.Pause;
   #Aux_OS := #_w1;
   "T10 LANT".Memory."Local StopAuto" := (#Aux_OS AND NOT "T10 LANT".Memory."Local StopAuto") OR ("T10 LANT".Memory."Local StopAuto" AND NOT #Aux_OS);
END_REGION

REGION Network 25: From step 8 to step 14
   RUNG wire#powerrail
      Contact( "T10 LANT".Memory.MEM_PT_END )
      wire#w1
      Contact( "T10 LANT".Memory.TRK_PIPE_IN )
      Coil( "T10 LANT".Memory."S8->S14" )
   END_RUNG
   RUNG wire#powerrail
      Contact( "T10 LANT".Memory.C_E )
      Contact( "T10 LANT".Memory.Pas_Decel_Lant_T10 )
      I_Contact( "T10 LANT".Memory.Pas_Stop_Lant_T10 )
   END_RUNG wire#w1
   // the same network as SCL:
   "T10 LANT".Memory."S8->S14" := ("T10 LANT".Memory.MEM_PT_END OR ("T10 LANT".Memory.C_E AND "T10 LANT".Memory.Pas_Decel_Lant_T10 AND NOT "T10 LANT".Memory.Pas_Stop_Lant_T10)) AND "T10 LANT".Memory.TRK_PIPE_IN;
END_REGION

REGION Network 26: From step 10 to step 14
   RUNG wire#powerrail
      Contact( "T10 LANT".Memory.MEM_PT_END )
      wire#w1
      Contact( "T10 LANT".Memory.TRK_PIPE_IN )
      Coil( "T10 LANT".Memory."S10->S14" )
   END_RUNG
   RUNG wire#powerrail
      Contact( "T10 LANT".Memory.C_E )
      Contact( "T10 LANT".Memory.Pas_Decel_Lant_T10 )
   END_RUNG wire#w1
   // the same network as SCL:
   "T10 LANT".Memory."S10->S14" := ("T10 LANT".Memory.MEM_PT_END OR ("T10 LANT".Memory.C_E AND "T10 LANT".Memory.Pas_Decel_Lant_T10)) AND "T10 LANT".Memory.TRK_PIPE_IN;
END_REGION

REGION Network 27: From step 12 to step 3
   RUNG wire#powerrail
      I_Contact( "T10 LANT".Memory.C_TO )
      I_Contact( "T10 LANT".Memory.C_F )
      I_Contact( "T10 LANT".Memory.C_E )
      wire#w1
      I_Contact( "T10 LANT".Memory.MEM_PT_END )
      I_Contact( "T10 LANT".Memory.PT_END )
      wire#w2
      Coil( "T10 LANT".Memory."S12->S3" )
   END_RUNG
   RUNG wire#powerrail
      Contact( "T10 LANT".Memory.C_TO )
      I_Contact( "T10 LANT".Memory.Doi_Pasi )
   END_RUNG wire#w1
   RUNG wire#powerrail
      Contact( "T10 LANT".Memory.C_F )
      wire#w3
      Contact( "T10 LANT".Memory.PIPE_TO_CHARGE )
   END_RUNG wire#w2
   RUNG wire#powerrail
      Contact( "T10 LANT".Memory.C_E )
   END_RUNG wire#w3
   RUNG wire#powerrail
      Contact( "T10 LANT".Memory.C_TO )
      Contact( "T10 LANT".Memory.Doi_Pasi )
   END_RUNG wire#w3
   RUNG wire#w3
      I_Contact( "T10 LANT".Memory.PIPE_TO_CHARGE )
      wire#w4
      I_Contact( "T10 OPRITOR SEQ"."S03_Check Piece Presence".X )
   END_RUNG wire#w2
   RUNG wire#w4
      I_Contact( "T10 OPRITOR".Memory.UP )
   END_RUNG wire#w2
   // the same network as SCL:
   "T10 LANT".Memory."S12->S3" := (((NOT "T10 LANT".Memory.C_TO AND NOT "T10 LANT".Memory.C_F AND NOT "T10 LANT".Memory.C_E) OR ("T10 LANT".Memory.C_TO AND NOT "T10 LANT".Memory.Doi_Pasi)) AND NOT "T10 LANT".Memory.MEM_PT_END AND NOT "T10 LANT".Memory.PT_END) OR (("T10 LANT".Memory.C_F OR "T10 LANT".Memory.C_E OR ("T10 LANT".Memory.C_TO AND "T10 LANT".Memory.Doi_Pasi)) AND ("T10 LANT".Memory.PIPE_TO_CHARGE OR (NOT "T10 LANT".Memory.PIPE_TO_CHARGE AND (NOT "T10 OPRITOR SEQ"."S03_Check Piece Presence".X OR NOT "T10 OPRITOR".Memory.UP))));
END_REGION

REGION Network 28: From step 12 to step 8
   RUNG wire#powerrail
      Contact( "T10 LANT".Memory.C_F )
      wire#w1
      I_Contact( "T10 LANT".Memory.PIPE_TO_CHARGE )
      wire#w2
      Contact( "T10 OPRITOR SEQ"."S03_Check Piece Presence".X )
      Contact( "T10 OPRITOR".Memory.UP )
      I_Contact( "T10 LANT".Memory.PT_END )
      I_Contact( "T10 LANT".Memory.MEM_PT_END )
      wire#w3
      Coil( "T10 LANT".Memory."S12->S8" )
   END_RUNG
   RUNG wire#powerrail
      Contact( "T10 LANT".Memory.C_E )
   END_RUNG wire#w1
   RUNG wire#powerrail
      Contact( "T10 LANT".Memory.C_TO )
      Contact( "T10 LANT".Memory.Doi_Pasi )
   END_RUNG wire#w1
   RUNG wire#w2
      I_Contact( "T10 LANT".Memory.PT_RALL )
      I_Contact( "T10 LANT".Memory.TRK_PIPE_LAST )
   END_RUNG wire#w3
   // the same network as SCL:
   "T10 LANT".Memory."S12->S8" := ("T10 LANT".Memory.C_F OR "T10 LANT".Memory.C_E OR ("T10 LANT".Memory.C_TO AND "T10 LANT".Memory.Doi_Pasi)) AND NOT "T10 LANT".Memory.PIPE_TO_CHARGE AND (("T10 OPRITOR SEQ"."S03_Check Piece Presence".X AND "T10 OPRITOR".Memory.UP AND NOT "T10 LANT".Memory.PT_END AND NOT "T10 LANT".Memory.MEM_PT_END) OR (NOT "T10 LANT".Memory.PT_RALL AND NOT "T10 LANT".Memory.TRK_PIPE_LAST));
END_REGION

REGION Network 29: From step 12 to step 14
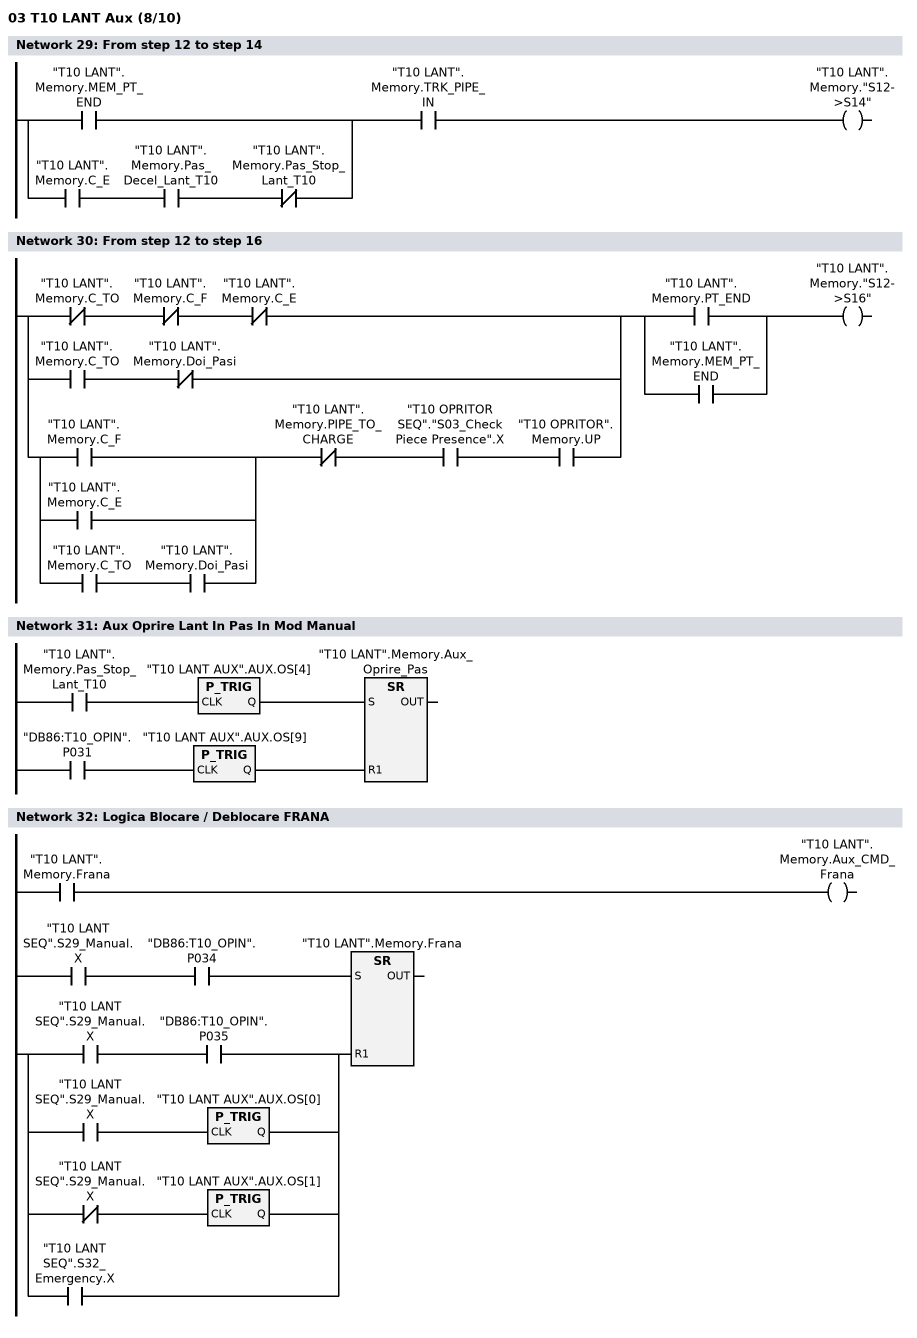
   RUNG wire#powerrail
      Contact( "T10 LANT".Memory.MEM_PT_END )
      wire#w1
      Contact( "T10 LANT".Memory.TRK_PIPE_IN )
      Coil( "T10 LANT".Memory."S12->S14" )
   END_RUNG
   RUNG wire#powerrail
      Contact( "T10 LANT".Memory.C_E )
      Contact( "T10 LANT".Memory.Pas_Decel_Lant_T10 )
      I_Contact( "T10 LANT".Memory.Pas_Stop_Lant_T10 )
   END_RUNG wire#w1
   // the same network as SCL:
   "T10 LANT".Memory."S12->S14" := ("T10 LANT".Memory.MEM_PT_END OR ("T10 LANT".Memory.C_E AND "T10 LANT".Memory.Pas_Decel_Lant_T10 AND NOT "T10 LANT".Memory.Pas_Stop_Lant_T10)) AND "T10 LANT".Memory.TRK_PIPE_IN;
END_REGION

REGION Network 30: From step 12 to step 16
   RUNG wire#powerrail
      I_Contact( "T10 LANT".Memory.C_TO )
      I_Contact( "T10 LANT".Memory.C_F )
      I_Contact( "T10 LANT".Memory.C_E )
      wire#w1
      Contact( "T10 LANT".Memory.PT_END )
      wire#w3
      Coil( "T10 LANT".Memory."S12->S16" )
   END_RUNG
   RUNG wire#powerrail
      Contact( "T10 LANT".Memory.C_TO )
      I_Contact( "T10 LANT".Memory.Doi_Pasi )
   END_RUNG wire#w1
   RUNG wire#powerrail
      Contact( "T10 LANT".Memory.C_F )
      wire#w2
      I_Contact( "T10 LANT".Memory.PIPE_TO_CHARGE )
      Contact( "T10 OPRITOR SEQ"."S03_Check Piece Presence".X )
      Contact( "T10 OPRITOR".Memory.UP )
   END_RUNG wire#w1
   RUNG wire#powerrail
      Contact( "T10 LANT".Memory.C_E )
   END_RUNG wire#w2
   RUNG wire#powerrail
      Contact( "T10 LANT".Memory.C_TO )
      Contact( "T10 LANT".Memory.Doi_Pasi )
   END_RUNG wire#w2
   RUNG wire#w1
      Contact( "T10 LANT".Memory.MEM_PT_END )
   END_RUNG wire#w3
   // the same network as SCL:
   "T10 LANT".Memory."S12->S16" := ((NOT "T10 LANT".Memory.C_TO AND NOT "T10 LANT".Memory.C_F AND NOT "T10 LANT".Memory.C_E) OR ("T10 LANT".Memory.C_TO AND NOT "T10 LANT".Memory.Doi_Pasi) OR (("T10 LANT".Memory.C_F OR "T10 LANT".Memory.C_E OR ("T10 LANT".Memory.C_TO AND "T10 LANT".Memory.Doi_Pasi)) AND NOT "T10 LANT".Memory.PIPE_TO_CHARGE AND "T10 OPRITOR SEQ"."S03_Check Piece Presence".X AND "T10 OPRITOR".Memory.UP)) AND ("T10 LANT".Memory.PT_END OR "T10 LANT".Memory.MEM_PT_END);
END_REGION

REGION Network 31: Aux Oprire Lant In Pas In Mod Manual
   RUNG wire#powerrail
      Contact( "T10 LANT".Memory.Pas_Stop_Lant_T10 )
      P_Trig( "T10 LANT AUX".AUX.OS[4] )
      S_SR(operand := "T10 LANT".Memory.Aux_Oprire_Pas, r1 := wire#w1)
   END_RUNG
   RUNG wire#powerrail
      Contact( "DB86:T10_OPIN".P031 )
      P_Trig( "T10 LANT AUX".AUX.OS[9] )
   END_RUNG wire#w1
   // the same network as SCL:
   #_w1 := "T10 LANT".Memory.Pas_Stop_Lant_T10 AND NOT "T10 LANT AUX".AUX.OS[4];   // rising edge
   "T10 LANT AUX".AUX.OS[4] := "T10 LANT".Memory.Pas_Stop_Lant_T10;
   #_w2 := "DB86:T10_OPIN".P031 AND NOT "T10 LANT AUX".AUX.OS[9];   // rising edge
   "T10 LANT AUX".AUX.OS[9] := "DB86:T10_OPIN".P031;
   IF #_w1 THEN
       "T10 LANT".Memory.Aux_Oprire_Pas := TRUE;   // SR flip-flop
   END_IF;
   IF #_w2 THEN "T10 LANT".Memory.Aux_Oprire_Pas := FALSE; END_IF;
END_REGION

REGION Network 32: Logica Blocare / Deblocare FRANA
   RUNG wire#powerrail
      Contact( "T10 LANT".Memory.Frana )
      Coil( "T10 LANT".Memory.Aux_CMD_Frana )
   END_RUNG
   RUNG wire#powerrail
      Contact( "T10 LANT SEQ".S29_Manual.X )
      Contact( "DB86:T10_OPIN".P034 )
      S_SR(operand := "T10 LANT".Memory.Frana, r1 := wire#w1)
   END_RUNG
   RUNG wire#powerrail
      Contact( "T10 LANT SEQ".S29_Manual.X )
      Contact( "DB86:T10_OPIN".P035 )
   END_RUNG wire#w1
   RUNG wire#powerrail
      Contact( "T10 LANT SEQ".S29_Manual.X )
      P_Trig( "T10 LANT AUX".AUX.OS[0] )
   END_RUNG wire#w1
   RUNG wire#powerrail
      I_Contact( "T10 LANT SEQ".S29_Manual.X )
      P_Trig( "T10 LANT AUX".AUX.OS[1] )
   END_RUNG wire#w1
   RUNG wire#powerrail
      Contact( "T10 LANT SEQ".S32_Emergency.X )
   END_RUNG wire#w1
   // the same network as SCL:
   "T10 LANT".Memory.Aux_CMD_Frana := "T10 LANT".Memory.Frana;
   #_w1 := "T10 LANT SEQ".S29_Manual.X AND NOT "T10 LANT AUX".AUX.OS[0];   // rising edge
   "T10 LANT AUX".AUX.OS[0] := "T10 LANT SEQ".S29_Manual.X;
   #_w2 := NOT "T10 LANT SEQ".S29_Manual.X AND NOT "T10 LANT AUX".AUX.OS[1];   // rising edge
   "T10 LANT AUX".AUX.OS[1] := NOT "T10 LANT SEQ".S29_Manual.X;
   IF "T10 LANT SEQ".S29_Manual.X AND "DB86:T10_OPIN".P034 THEN
       "T10 LANT".Memory.Frana := TRUE;   // SR flip-flop
   END_IF;
   IF ("T10 LANT SEQ".S29_Manual.X AND "DB86:T10_OPIN".P035) OR #_w1 OR #_w2 OR "T10 LANT SEQ".S32_Emergency.X THEN
       "T10 LANT".Memory.Frana := FALSE;
   END_IF;
END_REGION

REGION Network 33: ============= LENGHT MEASUREMENT =============
END_REGION

REGION Network 34: Encoder Preset
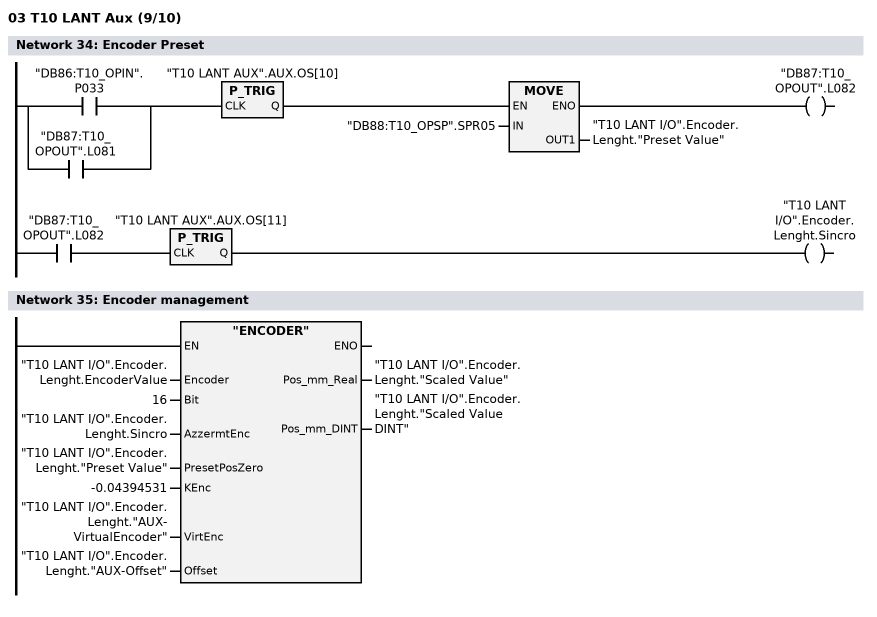
   RUNG wire#powerrail
      Contact( "DB86:T10_OPIN".P033 )
      wire#w1
      P_Trig( "T10 LANT AUX".AUX.OS[10] )
      Move(in := "DB88:T10_OPSP".SPR05, out1 => "T10 LANT I/O".Encoder.Lenght."Preset Value")
      Coil( "DB87:T10_OPOUT".L082 )
   END_RUNG
   RUNG wire#powerrail
      Contact( "DB87:T10_OPOUT".L081 )
   END_RUNG wire#w1
   RUNG wire#powerrail
      Contact( "DB87:T10_OPOUT".L082 )
      P_Trig( "T10 LANT AUX".AUX.OS[11] )
      Coil( "T10 LANT I/O".Encoder.Lenght.Sincro )
   END_RUNG
   // the same network as SCL:
   #_w1 := "DB86:T10_OPIN".P033 OR "DB87:T10_OPOUT".L081;
   #_w2 := #_w1 AND NOT "T10 LANT AUX".AUX.OS[10];   // rising edge
   "T10 LANT AUX".AUX.OS[10] := #_w1;
   IF #_w2 THEN "T10 LANT I/O".Encoder.Lenght."Preset Value" := "DB88:T10_OPSP".SPR05; END_IF;
   "DB87:T10_OPOUT".L082 := #_w2;
   #_w3 := "DB87:T10_OPOUT".L082 AND NOT "T10 LANT AUX".AUX.OS[11];   // rising edge
   "T10 LANT AUX".AUX.OS[11] := "DB87:T10_OPOUT".L082;
   "T10 LANT I/O".Encoder.Lenght.Sincro := #_w3;
END_REGION

REGION Network 35: Encoder management
   RUNG wire#powerrail
      "ENCODER"(Encoder := "T10 LANT I/O".Encoder.Lenght.EncoderValue, Bit := 16, AzzermtEnc := "T10 LANT I/O".Encoder.Lenght.Sincro, PresetPosZero := "T10 LANT I/O".Encoder.Lenght."Preset Value", KEnc := -0.04394531, VirtEnc := "T10 LANT I/O".Encoder.Lenght."AUX-VirtualEncoder", Offset := "T10 LANT I/O".Encoder.Lenght."AUX-Offset", Pos_mm_Real => "T10 LANT I/O".Encoder.Lenght."Scaled Value", Pos_mm_DINT => "T10 LANT I/O".Encoder.Lenght."Scaled Value DINT")
   END_RUNG
   // the same network as SCL:
   "ENCODER"(Encoder := "T10 LANT I/O".Encoder.Lenght.EncoderValue,
             Bit := 16,
             AzzermtEnc := "T10 LANT I/O".Encoder.Lenght.Sincro,
             PresetPosZero := "T10 LANT I/O".Encoder.Lenght."Preset Value",
             KEnc := -0.04394531,
             VirtEnc := "T10 LANT I/O".Encoder.Lenght."AUX-VirtualEncoder",
             Offset := "T10 LANT I/O".Encoder.Lenght."AUX-Offset",
             Pos_mm_Real => "T10 LANT I/O".Encoder.Lenght."Scaled Value",
             Pos_mm_DINT => "T10 LANT I/O".Encoder.Lenght."Scaled Value DINT");
END_REGION

REGION Network 36: Encoder 360
   // Calculeaza in functie de pozitia dorita 
   // 1. SetposOK = 110.0 (Treshhold = 10.0) (0.0 -> 340.0 viteza mare)
   //                                       340.0 -> 350.0 Viteza mica
   //                                       350.0 -> 360.0 Inertie oprire)
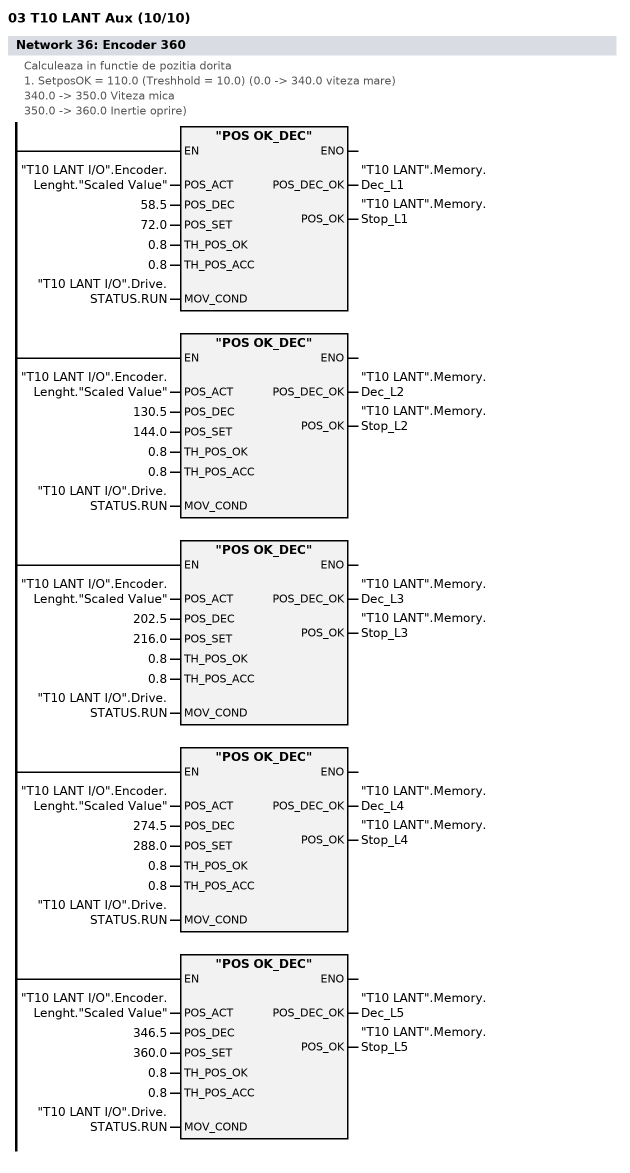
   RUNG wire#powerrail
      "POS OK_DEC"(POS_ACT := "T10 LANT I/O".Encoder.Lenght."Scaled Value", POS_DEC := 58.5, POS_SET := 72.0, TH_POS_OK := 0.8, TH_POS_ACC := 0.8, MOV_COND := "T10 LANT I/O".Drive.STATUS.RUN, POS_DEC_OK => "T10 LANT".Memory.Dec_L1, POS_OK => "T10 LANT".Memory.Stop_L1)
   END_RUNG
   RUNG wire#powerrail
      "POS OK_DEC"(POS_ACT := "T10 LANT I/O".Encoder.Lenght."Scaled Value", POS_DEC := 130.5, POS_SET := 144.0, TH_POS_OK := 0.8, TH_POS_ACC := 0.8, MOV_COND := "T10 LANT I/O".Drive.STATUS.RUN, POS_DEC_OK => "T10 LANT".Memory.Dec_L2, POS_OK => "T10 LANT".Memory.Stop_L2)
   END_RUNG
   RUNG wire#powerrail
      "POS OK_DEC"(POS_ACT := "T10 LANT I/O".Encoder.Lenght."Scaled Value", POS_DEC := 202.5, POS_SET := 216.0, TH_POS_OK := 0.8, TH_POS_ACC := 0.8, MOV_COND := "T10 LANT I/O".Drive.STATUS.RUN, POS_DEC_OK => "T10 LANT".Memory.Dec_L3, POS_OK => "T10 LANT".Memory.Stop_L3)
   END_RUNG
   RUNG wire#powerrail
      "POS OK_DEC"(POS_ACT := "T10 LANT I/O".Encoder.Lenght."Scaled Value", POS_DEC := 274.5, POS_SET := 288.0, TH_POS_OK := 0.8, TH_POS_ACC := 0.8, MOV_COND := "T10 LANT I/O".Drive.STATUS.RUN, POS_DEC_OK => "T10 LANT".Memory.Dec_L4, POS_OK => "T10 LANT".Memory.Stop_L4)
   END_RUNG
   RUNG wire#powerrail
      "POS OK_DEC"(POS_ACT := "T10 LANT I/O".Encoder.Lenght."Scaled Value", POS_DEC := 346.5, POS_SET := 360.0, TH_POS_OK := 0.8, TH_POS_ACC := 0.8, MOV_COND := "T10 LANT I/O".Drive.STATUS.RUN, POS_DEC_OK => "T10 LANT".Memory.Dec_L5, POS_OK => "T10 LANT".Memory.Stop_L5)
   END_RUNG
   // the same network as SCL:
   "POS OK_DEC"(POS_ACT := "T10 LANT I/O".Encoder.Lenght."Scaled Value",
                POS_DEC := 58.5,
                POS_SET := 72.0,
                TH_POS_OK := 0.8,
                TH_POS_ACC := 0.8,
                MOV_COND := "T10 LANT I/O".Drive.STATUS.RUN,
                POS_DEC_OK => "T10 LANT".Memory.Dec_L1,
                POS_OK => "T10 LANT".Memory.Stop_L1);
   "POS OK_DEC"(POS_ACT := "T10 LANT I/O".Encoder.Lenght."Scaled Value",
                POS_DEC := 130.5,
                POS_SET := 144.0,
                TH_POS_OK := 0.8,
                TH_POS_ACC := 0.8,
                MOV_COND := "T10 LANT I/O".Drive.STATUS.RUN,
                POS_DEC_OK => "T10 LANT".Memory.Dec_L2,
                POS_OK => "T10 LANT".Memory.Stop_L2);
   "POS OK_DEC"(POS_ACT := "T10 LANT I/O".Encoder.Lenght."Scaled Value",
                POS_DEC := 202.5,
                POS_SET := 216.0,
                TH_POS_OK := 0.8,
                TH_POS_ACC := 0.8,
                MOV_COND := "T10 LANT I/O".Drive.STATUS.RUN,
                POS_DEC_OK => "T10 LANT".Memory.Dec_L3,
                POS_OK => "T10 LANT".Memory.Stop_L3);
   "POS OK_DEC"(POS_ACT := "T10 LANT I/O".Encoder.Lenght."Scaled Value",
                POS_DEC := 274.5,
                POS_SET := 288.0,
                TH_POS_OK := 0.8,
                TH_POS_ACC := 0.8,
                MOV_COND := "T10 LANT I/O".Drive.STATUS.RUN,
                POS_DEC_OK => "T10 LANT".Memory.Dec_L4,
                POS_OK => "T10 LANT".Memory.Stop_L4);
   "POS OK_DEC"(POS_ACT := "T10 LANT I/O".Encoder.Lenght."Scaled Value",
                POS_DEC := 346.5,
                POS_SET := 360.0,
                TH_POS_OK := 0.8,
                TH_POS_ACC := 0.8,
                MOV_COND := "T10 LANT I/O".Drive.STATUS.RUN,
                POS_DEC_OK => "T10 LANT".Memory.Dec_L5,
                POS_OK => "T10 LANT".Memory.Stop_L5);
END_REGION
END_FUNCTION
